// TIA Portal V19 export
TYPE "OOAx_Config"
// stored: Access Published
   STRUCT
      limitMinus : LReal;   // Par: software limit in minus direction [unit] / mm
      limitPlus : LReal;   // Par: software limit in minus direction [unit] / mm
      Backlash : LReal;   // mm
      BacklashActivation : Bool;
      ToleranceWindow : LReal;   // mm
      ToleranceWindowDelay : Time;
      PreCutOff : LReal;   // mm
      PreEndLowSpeed : LReal;   // mm
      PreEndMedSpeed : LReal;   // mm
      ChangeDirectionDelay : Time;
      StandstillVelocity : LReal;   // xxxx : Depend from VelocityMeasUnit
      StandStillDelay : Time;
      HomingDirection : Bool;   // FALSE=Minus, TRUE=Plus
      RecallTime : LReal;   // Time for calculate speed in ms
      VelocityFilter_T : LReal := 10.0;   // Velocity filter time in ms
      VelocityMeasUnit : Int;   // 0=m/min, 1=m/s, 2=mm/s
      PosFbkDisabled : Bool;   // PosFbk is disbled (only Jog Command)
      FbkCtrlDisabled : Bool;   // Disable controls of feedback behaviour
   END_STRUCT;
END_TYPE
